FUNCTION_BLOCK WTAV_UINT (* Weighted Average *)
  (* Standard: 61499-1; Classification: Math; Function: Weighted average *)
  (* Version 0.5, 2008-06-27, JHC, Holobloc Inc, Redefined IN1, IN2 to parallel WTAV_PCT; subclassed from FBFunction2. *)
  (* Version 0.4, 2005-06-01, JHC, Holobloc Inc, Re-compiled with new emitter. *)
  (* Version 0.3, 2004-09-25, JHC, Rockwell Automation, Deleted INIT, INITO; moved to fb.rt.math. *)
  (* Version 0.2, 2003-03-17, JHC, Rockwell Automation, Moved from fb.rt.omac to fb.rt.mach. *)
  (* Version 0.1, 2002-02-28, JHC, Rockwell Automation, Changed "=" to ":=", REAL_TO_INT to Java cast in ALGORITHM REQ. *)
  (* Version 0.0, 2001-04-14, JHC, Rockwell Automation, First XML version *)
  (* Compiler header: package fb.rt.math; *)
  (* Compiler classdef: public class WTAV_UINT extends FBFunction2 *)
  (* Compiler Java Sun JDK 1.6.0 *)
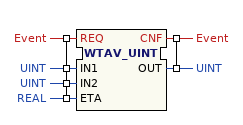
  EVENT_INPUT
    REQ WITH IN1, IN2, ETA; (* Normal Calculation *)
  END_EVENT
  EVENT_OUTPUT
    CNF WITH OUT; (* Execution Confirmation *)
  END_EVENT
  VAR_INPUT
    IN1 : UINT; (* Value when ETA=0.0 *)
    IN2 : UINT; (* Value when ETA=1.0 *)
    ETA : REAL; (* Weighting factor, internally limited to (0.0..1.0) *)
  END_VAR
  VAR_OUTPUT
    OUT : UINT; (* ETA*X1+(1-ETA)*X2 *)
  END_VAR
END_FUNCTION_BLOCK
